// TIA Portal V18 export
// export: Created 2025-12-01T17:51:31.0261906Z, ExportSetting None, DisplayName Totally Integrated Automation Portal, DisplayVersion V18 Update 5, DisplayName TIA Portal Openness, DisplayVersion V18 Update 5, DisplayName TIA Portal Teamcenter Gateway, DisplayVersion V18, DisplayName TIA Portal Version Control Interface, DisplayVersion V18, DisplayName STEP 7 Professional, DisplayVersion V18 Update 5, DisplayName STEP 7 Safety, DisplayVersion V18, DisplayName WinCC Professional, DisplayVersion V18 Update 5
DATA_BLOCK "DB_Commissioning"   // DB32767
{ S7_Optimized_Access := 'TRUE' }
// stored: AutoNumber false, MemoryReserve 100
   VAR RETAIN
      str : Array[1..8] of String[60];
      bit : Array[1..8] of Bool;
   END_VAR
BEGIN
   str[1] := 'LE4B171420124M33700000131950710';
END_DATA_BLOCK
